// TIA Portal V19 export
TYPE "PPrf_CoilHandlig"
// stored: Access Published
   STRUCT
      MaterialFeeding : "PPrf_CoilHandling_MaterialFeeding";
      WeldingCycle { S7_SetPoint := 'True'} : "PPrf_CoilHandling_WeldingCycle";
   END_STRUCT;
END_TYPE
